INTERFACE ITF_Component_TE1_HMI EXTENDS ITF_BaseComponent_HMI

METHOD LinkComponentData : BOOL
VAR_INPUT
	stData				: REFERENCE TO ST_Component_TE1_HMI_Link;
END_VAR
END_METHOD

END_INTERFACE

(* stored: Version 1.1.0.1, ProductVersion 3.1.4024.15
   Itf ITF_Component_TE1_HMI: Id {65d00de8-2314-46c2-9637-ac9cd2e82de8}
   Method LinkComponentData: Id {d3389f5d-0e11-434d-8b5a-8e0f1693584e} *)
